KUKA KRL data list: braketestreq.dat

&ACCESS RVO1
&COMMENT BrkTst-main task
&PARAM DISKPATH = KRC:\R1\TP\BrakeTest
&PARAM EDITMASK = *
DEFDAT  BRAKETESTREQ PUBLIC
;FOLD EXTERNAL DECLARATIONS;%{PE}%MKUKATPBASIS,%CEXT,%VCOMMON,%P
;FOLD GRIPPERTECH EXT
  EXT  H50 (INT:IN, INT:IN ,INT:IN ,GRP_TYP:IN)
;ENDFOLD (GRIPPERTECH EXT)
;FOLD SPOTTECH EXT
  EXT  USERSPOT (S_COMMAND  :IN, SPOT_TYPE:IN)
;ENDFOLD (SPOTTECH EXT)
;FOLD BASISTECH EXT;%{PE}%MKUKATPBASIS,%CEXT,%VEXT,%P
DECL INT SUCCESS
;ENDFOLD (BASISTECH EXT)
;FOLD USER EXT;%{E}%MKUKATPUSER,%CEXT,%VEXT,%P
;ENDFOLD (USER EXT)
;ENDFOLD (EXTERNAL DECLERATIONS)

; The name of the brake test device as in in motiondrv.ini
GLOBAL CHAR brakeTestDevName[30]
brakeTestDevName[]="BRAKE_TEST"

GLOBAL CHAR brakeTestMdbName[30]
brakeTestMdbName[]="BrkTst"

INT AxNr,BtIrNr

ENDDAT
